TYPE ST_TEST_SETTING :
STRUCT
	height:		UDINT;
	width:		UDINT;
	x:			UDINT;
	y:			UDINT;
END_STRUCT
END_TYPE

(* stored: Version 1.1.0.1
   DUT ST_TEST_SETTING: Id {271dd325-0fd1-457e-b4be-58284892e23e} *)
